Staubli VAL3: WacohFTSensor2.dtx

public bool bOverRun = true
mdesc mNomSpeed
public num nForceTorque[6]
  [0] = -0.458435
  [1] = -0.0611247
  [2] = -0.0305157
  [3] = 0.00182448
  [4] = 0.00243784
public num nPort = 5001
public num nSensitivity[6]
  [0] = 32.72
  [1] = 32.72
  [2] = 32.77
  [3] = 1644.3
  [4] = 1640.8
  [5] = 1635
public num nSioTimeOut = 5
public num nZeroPoint[6]
  [0] = 8211
  [1] = 8189
  [2] = 8176
  [3] = 8194
  [4] = 8176
  [5] = 8189
public sio sClient = {link=Socket\FTSensor}
